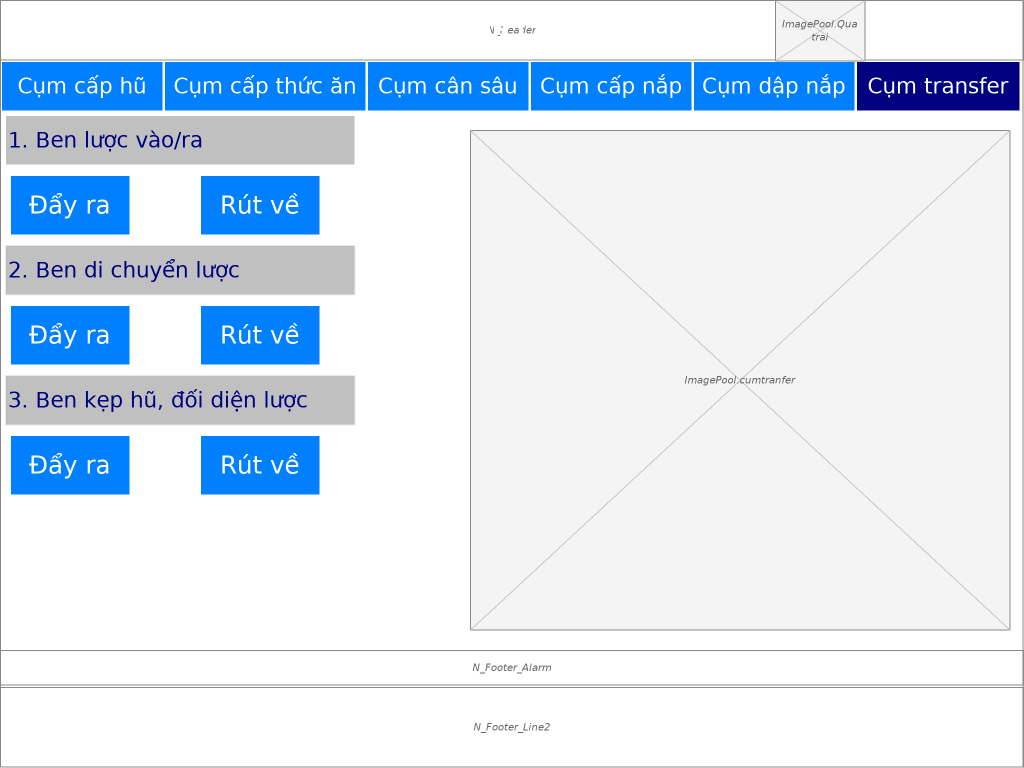
VISUALIZATION N_Tranfer2  // 1024x768
    Rectangle (10,305 120x60), "Đẩy ra", colour toggle: PR_Line02.bCylinder_Move_Comb_Extend, input disabled if: Not PR_Line02.bCheck
        OnMouseDown: execute { PR_Line02.bCylinder_Move_Comb_Extend := TRUE; PR_Line02.bCylinder_Move_Comb_Retract := FALSE; }
    Rectangle (200,175 120x60), "Rút về", colour toggle: PR_Line02.bCylinder_Comb_Retract
        OnMouseDown: execute { PR_Line02.bCylinder_Comb_Retract := TRUE; PR_Line02.bCylinder_Comb_Extend := FALSE; }
    Rectangle (200,305 120x60), "Rút về", colour toggle: PR_Line02.bCylinder_Move_Comb_Retract, input disabled if: Not PR_Line02.bCheck
        OnMouseDown: execute { PR_Line02.bCylinder_Move_Comb_Retract := TRUE; PR_Line02.bCylinder_Move_Comb_Extend := FALSE; }
    Frame (0,687 1024x80)
        shows N_Footer_Line2()
    Frame (0,0 1024x60)
        shows N_Header()
    Textfield (353,5 400x50), "MÀN HÌNH CHẠY TAY LINE 2"
    Rectangle (10,175 120x60), "Đẩy ra", colour toggle: PR_Line02.bCylinder_Comb_Extend, input disabled if: Not PR_Line02.bCheck
        OnMouseDown: execute { PR_Line02.bCylinder_Comb_Extend := TRUE; PR_Line02.bCylinder_Comb_Retract := FALSE; }
    Rectangle (1,61 162x50), "Cụm cấp hũ"
        OnMouseClick: change screen: N_JarSupply2
    Rectangle (164,61 202x50), "Cụm cấp thức ăn"
        OnMouseClick: change screen: N_FoodSupply2
    Rectangle (367,61 162x50), "Cụm cân sâu"
        OnMouseClick: change screen: N_WormWeight2
    Rectangle (530,61 162x50), "Cụm cấp nắp"
        OnMouseClick: change screen: N_LidSupply2
    Rectangle (693,61 162x50), "Cụm dập nắp"
        OnMouseClick: change screen: N_LidPressing2
    Rectangle (856,61 164x50), "Cụm transfer"
        OnMouseClick: change screen: N_Tranfer2
    Rectangle (200,435 120x60), "Rút về", colour toggle: PR_Line02.bCylinder_Clip_Retract
        OnMouseDown: execute { PR_Line02.bCylinder_Clip_Retract := TRUE; PR_Line02.bCylinder_Clip_Extend := FALSE; }
    Rectangle (10,435 120x60), "Đẩy ra", colour toggle: PR_Line02.bCylinder_Clip_Extend
        OnMouseDown: execute { PR_Line02.bCylinder_Clip_Extend := TRUE; PR_Line02.bCylinder_Clip_Retract := FALSE; }
    Image (775,0 90x61), input disabled if: bResetAuto1, image: ImagePool.Qua trai
        OnMouseClick: change screen: N_Tranfer1
        OnMouseClick: execute { MAIN.bModeManual := TRUE; MAIN.bModeAuto := FALSE; }
    Rectangle (5,115 350x50), "1. Ben lược vào/ra"
    Rectangle (5,245 350x50), "2. Ben di chuyển lược"
    Rectangle (5,375 350x50), "3. Ben kẹp hũ, đối diện lược"
    Image (470,130 540x500), image: ImagePool.cumtranfer
    Frame (0,650 1024x35)
        shows N_Footer_Alarm()
END_VISUALIZATION

(* stored: Version 1.1.0.1, ProductVersion 3.1.4024.12
   Visu N_Tranfer2: Id {b915c630-b697-4781-8163-18f6b62a58a9} *)
